(* PLC project marvel_dome, Institute of Astronomy Onto 0.0.1 *)
(* stored: creationDateTime 2025-02-14T19:08:53.030329, modificationDateTime 2025-02-14T19:08:53.030329 *)

TYPE DomeShutterMotionStates : (STANDSTILL := 0, OPENING := 1, CLOSING := 2, STOPPING := 3, TIMEOUT_ERROR := 4, RETRY_OPENING := 5, RETRY_CLOSING := 6, UNKNOWN_DRIVE_LOGIC_ERROR := 7) BYTE;
END_TYPE

TYPE DomeShutterApertureStates : (UNKNOWN := 0, FULLY_OPEN := 1, PARTIALLY_OPEN := 2, FULLY_CLOSED := 3, INVALID := 4) BYTE;
END_TYPE

TYPE DomeShutterCommands : (NONE := 0, STOP := 1, CLOSE := 2, OPEN := 3, SET_HUMIDITY_LIMIT := 4, SET_HEARTBEAT_TIMEOUT := 5, SET_DRIVE_LOGIC := 6) BYTE;
END_TYPE

TYPE DomeShutterDriveLogic : (UNKNOWN := 0, EDGE_BASED := 1, LEVEL_BASED := 2) BYTE;
END_TYPE

TYPE DomeParts : STRUCT
  shutter : DomeShutter;  (* Shutter mechanism *)
  rotation : DomeRotation;  (* Rotation mechanism *)
END_STRUCT;
END_TYPE

TYPE DomeRotationParts : STRUCT
  motorAxis : AngularAxis;  (* Motor axis *)
  encoderAxis : AngularAxis;  (* Encoder axis *)
END_STRUCT;
END_TYPE

TYPE DomeProcesses : STRUCT
  initialize : Process;  (* Start initializing *)
  changeOperatingState : ChangeOperatingStateProcess;  (* Change the operating state (e.g. AUTO, MANUAL, ...) *)
  lock : Process;  (* Lock the cover *)
  unlock : Process;  (* Unlock the cover *)
  reset : Process;  (* Reset any errors *)
  powerOn : Process;  (* Power on the dome *)
  powerOff : Process;  (* Power off the dome *)
  syncWithAxes : Process;  (* Synchronize the dome once with the axes *)
  startTracking : Process;  (* Start tracking the axes *)
  stopTracking : Process;  (* Stop tracking the axes *)
  stop : Process;  (* Stop the rotation movement and/or tracking *)
  moveKnownPosition : DomeMoveKnownPositionProcess;  (* Move the dome to the given known position *)
END_STRUCT;
END_TYPE

TYPE DomeShutterProcesses : STRUCT
  open : Process;  (* Open both panels *)
  close : Process;  (* Close both panels *)
  stop : Process;  (* Stop the panels *)
END_STRUCT;
END_TYPE

TYPE DomeRotationProcesses : STRUCT
  reset : Process;  (* Reset errors *)
  stop : Process;  (* Stop the rotation *)
  moveAbsolute : DomeMoveProcess;  (* Move absolute *)
  moveRelative : DomeMoveProcess;  (* Move relative *)
  powerOn : Process;  (* Power on master and slave *)
  powerOff : Process;  (* Power off master and slave *)
END_STRUCT;
END_TYPE

TYPE DomeStatuses : STRUCT
  initializationStatus : InitializationStatus;
  healthStatus : HealthStatus;
  busyStatus : BusyStatus;
  operatingStatus : OperatingStatus;
  poweredStatus : PoweredStatus;
END_STRUCT;
END_TYPE

TYPE DomeShutterStatuses : STRUCT
  apertureStatus : ApertureStatus;  (* Combined aperture status (i.e. of both panels) *)
  motionStatus : DomeShutterOpeningStatus;  (* Motion status *)
  healthStatus : HealthStatus;  (* Health status *)
  busyStatus : BusyStatus;  (* Busy status *)
END_STRUCT;
END_TYPE

TYPE DomeRotationStatuses : STRUCT
  healthStatus : HealthStatus;  (* Health status *)
  busyStatus : BusyStatus;  (* Busy status *)
  poweredStatus : PoweredStatus;  (* Powered status *)
END_STRUCT;
END_TYPE

TYPE DomeConfig : STRUCT
  shutter : DomeShutterConfig;  (* The config of the shutter mechanism *)
  rotation : DomeRotationConfig;  (* The config of the rotation system *)
  maxTrackingDistance : LREAL;  (* The maximum distance between telescope and dome while tracking *)
  trackingLoopTime : LREAL;  (* Loop time, in seconds, of the tracking. *)
  knownPositions : DomeKnownPositionsConfig;  (* The known positions of the dome *)
  knownPositionTolerance : LREAL;  (* Tolerance (in degrees) to determine if the dome is at a known position *)
END_STRUCT;
END_TYPE

TYPE DomeKnownPositionConfig : STRUCT
  name : STRING;  (* The name of the position (e.g. 'PARK') *)
  position : LREAL;  (* Azimuth in degrees *)
END_STRUCT;
END_TYPE

TYPE DomeKnownPositionsConfig : STRUCT
  position0 : DomeKnownPositionConfig;  (* Known position 0 *)
  position1 : DomeKnownPositionConfig;  (* Known position 1 *)
  position2 : DomeKnownPositionConfig;  (* Known position 2 *)
  position3 : DomeKnownPositionConfig;  (* Known position 3 *)
  position4 : DomeKnownPositionConfig;  (* Known position 4 *)
  position5 : DomeKnownPositionConfig;  (* Known position 5 *)
  position6 : DomeKnownPositionConfig;  (* Known position 6 *)
  position7 : DomeKnownPositionConfig;  (* Known position 7 *)
  position8 : DomeKnownPositionConfig;  (* Known position 8 *)
  position9 : DomeKnownPositionConfig;  (* Known position 9 *)
END_STRUCT;
END_TYPE

TYPE DomeShutterConfig : STRUCT
  remotePlcAmsId : STRING;  (* AMS ID of the shutter PLC *)
  remotePlcTimeoutSeconds : LREAL;  (* The timeout of a single ADS command. *)
  simulated : BOOL := TRUE;  (* TRUE if the shutter is simulated, FALSE if not *)
  openingTimeoutSeconds : LREAL;  (* The opening timeout. *)
  closingTimeoutSeconds : LREAL;  (* The closing timeout. *)
END_STRUCT;
END_TYPE

TYPE DomeRotationConfig : STRUCT
  maxMovingVelocity : LREAL;  (* Maximum velocity when moving absolute or relative, in degrees per second *)
  maxMasterSlaveLag : LREAL;  (* Below this lag value (in degrees), the lag is considered not an error *)
  homePosition : LREAL;  (* Azimuth position of the home sensor, in degrees *)
END_STRUCT;
END_TYPE

{attribute 'pack_mode' := '8'}
TYPE DomeShutterDataRead : STRUCT
  motionState : DomeShutterMotionStates;  (* The motion state, as reported by the shutter PLC *)
  apertureState : DomeShutterApertureStates;  (* The aperture state, as reported by the shutter PLC *)
  heartBeatReceived : UDINT;  (* The heartbeat that was last received by the shutter PLC, as reported by the shutter PLC *)
  lastCommandReceived : DomeShutterCommands;  (* The command that was last received by the shutter PLC, as reported by the shutter PLC *)
  leftPanelOpen : BIT;  (* True if the left panel is open, False if not *)
  leftPanelClosed : BIT;  (* True if the left panel is closed, False if not *)
  rightPanelOpen : BIT;  (* True if the right panel is open, False if not *)
  rightPanelClosed : BIT;  (* True if the right panel is closed, False if not *)
  relayOpenActive : BIT;  (* True if the relay to open the shutter is active, False if not *)
  relayCloseActive : BIT;  (* True if the relay to close the shutter is active, False if not *)
  bHumidityUnderrange : BIT;  (* True if the humidity sensor is in underrange, False if not *)
  bHumidityOverrange : BIT;  (* True if the humidity sensor is in overrange, False if not *)
  bHumidityError : BIT;  (* True if the humidity sensor is in error, False if not *)
  bTemperatureUnderrange : BIT;  (* True if the temperature sensor is in underrange, False if not *)
  bTemperatureOverrange : BIT;  (* True if the temperature sensor is in overrange, False if not *)
  bTemperatureError : BIT;  (* True if the temperature sensor is in error, False if not *)
  heartBeatViolation : BIT;  (* True if there is a missing heartbeat reported by the shutter PLC, False if not *)
  humidityViolation : BIT;  (* True if there is high humidity reported by the shutter PLC, False if not *)
  driveLogic : DomeShutterDriveLogic;  (* Determines which logic is used by the shutter drives (edge or level based) *)
  humidityRawValue : INT;  (* The raw value of the humidity sensor *)
  temperatureRawValue : INT;  (* The raw value of the temperature sensor *)
  humidityLimit : INT;  (* Humidity limit (as raw sensor value) above which the dome will close automatically (-1 means turn off) *)
  heartBeatTimeout : INT;  (* Heartbeat timeout (in seconds) above which the dome will close automatically (-1 means turn off) *)
END_STRUCT;
END_TYPE

{attribute 'pack_mode' := '8'}
TYPE DomeShutterDataWrite : STRUCT
  heartBeat : UDINT;  (* The heartbeat to send to the shutter PLC *)
  command : DomeShutterCommands;  (* The command to send to the shutter PLC *)
  arg : INT;  (* The int16 argument belonging to the command (optional) *)
END_STRUCT;
END_TYPE

TYPE DomeMoveKnownPositionProcessArgs : STRUCT
  name : STRING;  (* Name of the position to move to *)
END_STRUCT;
END_TYPE

TYPE DomeMoveProcessArgs : STRUCT
  position : LREAL;  (* New absolute or relative position value in degrees *)
END_STRUCT;
END_TYPE

FUNCTION_BLOCK DomeShutterOpeningStatus
  VAR_INPUT
    superState : BOOL := TRUE;  (* Super state (TRUE if the super state is active, or if there is no super state) *)
    shutterValue : DomeShutterMotionStates;  (* Enum from mini PLC *)
  END_VAR
  VAR_OUTPUT
    {attribute 'OPC.UA.DA' := '1'}
    {attribute 'OPC.UA.DA.Access' := '1'}
    standstill : BOOL;  (* Standstill *)
    {attribute 'OPC.UA.DA' := '1'}
    {attribute 'OPC.UA.DA.Access' := '1'}
    opening : BOOL;  (* Opening *)
    {attribute 'OPC.UA.DA' := '1'}
    {attribute 'OPC.UA.DA.Access' := '1'}
    closing : BOOL;  (* Closing *)
    {attribute 'OPC.UA.DA' := '1'}
    {attribute 'OPC.UA.DA.Access' := '1'}
    stopping : BOOL;  (* Stopping *)
    {attribute 'OPC.UA.DA' := '1'}
    {attribute 'OPC.UA.DA.Access' := '1'}
    timeoutError : BOOL;  (* Timeout error *)
    {attribute 'OPC.UA.DA' := '1'}
    {attribute 'OPC.UA.DA.Access' := '1'}
    retryOpening : BOOL;  (* Retry opening *)
    {attribute 'OPC.UA.DA' := '1'}
    {attribute 'OPC.UA.DA.Access' := '1'}
    retryClosing : BOOL;  (* Retry closing *)
    {attribute 'OPC.UA.DA' := '1'}
    {attribute 'OPC.UA.DA.Access' := '1'}
    unknownDriveLogicError : BOOL;  (* Drive logic (edge based or dead-man switch) was not configured yet *)
  END_VAR

            standstill := (shutterValue = DomeShutterMotionStates.STANDSTILL) AND superState;
opening := (shutterValue = DomeShutterMotionStates.OPENING) AND superState;
closing := (shutterValue = DomeShutterMotionStates.CLOSING) AND superState;
stopping := (shutterValue = DomeShutterMotionStates.STOPPING) AND superState;
timeoutError := (shutterValue = DomeShutterMotionStates.TIMEOUT_ERROR) AND superState;
retryOpening := (shutterValue = DomeShutterMotionStates.RETRY_OPENING) AND superState;
retryClosing := (shutterValue = DomeShutterMotionStates.RETRY_CLOSING) AND superState;
unknownDriveLogicError := (shutterValue = DomeShutterMotionStates.UNKNOWN_DRIVE_LOGIC_ERROR) AND superState;

          
END_FUNCTION_BLOCK

FUNCTION_BLOCK SM_Dome
  VAR_OUTPUT
    {attribute 'OPC.UA.DA' := '1'}
    {attribute 'OPC.UA.DA.Access' := '1'}
    actualStatus : STRING;  (* Current status description *)
    previousStatus : STRING;  (* Previous status description *)
    {attribute 'OPC.UA.DA' := '1'}
    {attribute 'OPC.UA.DA.Access' := '1'}
    isTracking : BOOL;  (* True if the dome is tracking the telescope *)
    {attribute 'OPC.UA.DA' := '1'}
    {attribute 'OPC.UA.DA.Access' := '1'}
    isAtKnownPosition : BOOL;  (* True if the dome is at a known position *)
    {attribute 'OPC.UA.DA' := '1'}
    {attribute 'OPC.UA.DA.Access' := '1'}
    actualKnownPositionName : STRING;  (* Name of the known position if isAtKnownPosition is True *)
    statuses : DomeStatuses;  (* Statuses of the state machine *)
    parts : DomeParts;  (* Parts of the state machine *)
    processes : DomeProcesses;  (* Processes of the state machine *)
  END_VAR
  VAR_IN_OUT
    {attribute 'OPC.UA.DA' := '0'}
    operatorStatus : OperatorStatus;  (* Reference to the operator (observer/tech) *)
    {attribute 'OPC.UA.DA' := '0'}
    activityStatus : ActivityStatus;  (* Shared activity status *)
    {attribute 'OPC.UA.DA' := '0'}
    config : DomeConfig;  (* Active configuration of the cover *)
    {attribute 'OPC.UA.DA' := '0'}
    telescopeAzi : AngularPosition;  (* Azimuth target position of the telescope Axes *)
  END_VAR

            parts.shutter(
    initializationStatus := statuses.initializationStatus,
    operatorStatus := operatorStatus,
    operatingStatus := statuses.operatingStatus,
    activityStatus := activityStatus,
    config := config.shutter);
parts.rotation(
    initializationStatus := statuses.initializationStatus,
    operatorStatus := operatorStatus,
    operatingStatus := statuses.operatingStatus,
    config := config.rotation);
statuses.initializationStatus();
statuses.healthStatus(
    isGood := parts.shutter.statuses.healthStatus.isGood AND parts.rotation.statuses.healthStatus.isGood,
    hasWarning := parts.shutter.statuses.healthStatus.hasWarning OR parts.rotation.statuses.healthStatus.hasWarning);
statuses.busyStatus( isBusy := parts.shutter.statuses.busyStatus.busy OR parts.rotation.statuses.busyStatus.busy );
statuses.operatingStatus( superState := statuses.initializationStatus.initialized );
statuses.poweredStatus( isEnabled := parts.rotation.statuses.poweredStatus.enabled );
processes.initialize( isEnabled := (NOT(statuses.initializationStatus.locked)) AND (statuses.initializationStatus.shutdown OR (statuses.initializationStatus.initializingFailed OR statuses.initializationStatus.initialized)) );
processes.changeOperatingState( isEnabled := FALSE );
processes.lock( isEnabled := operatorStatus.tech );
processes.unlock( isEnabled := operatorStatus.tech AND statuses.initializationStatus.locked );
processes.reset( isEnabled := statuses.busyStatus.idle AND statuses.initializationStatus.initialized );
processes.powerOn( isEnabled := (NOT(statuses.initializationStatus.locked)) AND (statuses.initializationStatus.initialized AND processes.powerOn.statuses.busyStatus.idle) );
processes.powerOff( isEnabled := statuses.initializationStatus.initialized AND processes.powerOff.statuses.busyStatus.idle );
processes.syncWithAxes( isEnabled := statuses.initializationStatus.initialized AND (statuses.busyStatus.idle AND statuses.poweredStatus.enabled) );
processes.startTracking( isEnabled := statuses.poweredStatus.enabled AND (NOT(isTracking)) );
processes.stopTracking( isEnabled := isTracking );
processes.stop( isEnabled := statuses.busyStatus.busy OR (isTracking OR operatorStatus.tech) );
processes.moveKnownPosition( isEnabled := statuses.initializationStatus.initialized AND (statuses.busyStatus.idle AND statuses.poweredStatus.enabled) );

          

{attribute 'TcRpcEnable' := '1'}
METHOD initialize : RequestResults
                  initialize := THIS^.processes.initialize.request();

                
END_METHOD

{attribute 'TcRpcEnable' := '1'}
METHOD changeOperatingState : RequestResults
  VAR_INPUT
    state : OperatingStates;
  END_VAR
                  changeOperatingState := THIS^.processes.changeOperatingState.request( state := state );

                
END_METHOD

{attribute 'TcRpcEnable' := '1'}
METHOD lock : RequestResults
                  lock := THIS^.processes.lock.request();

                
END_METHOD

{attribute 'TcRpcEnable' := '1'}
METHOD unlock : RequestResults
                  unlock := THIS^.processes.unlock.request();

                
END_METHOD

{attribute 'TcRpcEnable' := '1'}
METHOD reset : RequestResults
                  reset := THIS^.processes.reset.request();

                
END_METHOD

{attribute 'TcRpcEnable' := '1'}
METHOD powerOn : RequestResults
                  powerOn := THIS^.processes.powerOn.request();

                
END_METHOD

{attribute 'TcRpcEnable' := '1'}
METHOD powerOff : RequestResults
                  powerOff := THIS^.processes.powerOff.request();

                
END_METHOD

{attribute 'TcRpcEnable' := '1'}
METHOD syncWithAxes : RequestResults
                  syncWithAxes := THIS^.processes.syncWithAxes.request();

                
END_METHOD

{attribute 'TcRpcEnable' := '1'}
METHOD startTracking : RequestResults
                  startTracking := THIS^.processes.startTracking.request();

                
END_METHOD

{attribute 'TcRpcEnable' := '1'}
METHOD stopTracking : RequestResults
                  stopTracking := THIS^.processes.stopTracking.request();

                
END_METHOD

{attribute 'TcRpcEnable' := '1'}
METHOD stop : RequestResults
                  stop := THIS^.processes.stop.request();

                
END_METHOD

{attribute 'TcRpcEnable' := '1'}
METHOD moveKnownPosition : RequestResults
  VAR_INPUT
    name : STRING;
  END_VAR
                  moveKnownPosition := THIS^.processes.moveKnownPosition.request( name := name );

                
END_METHOD

METHOD _log : BOOL
  VAR_INPUT
    name : STRING;  (* Name of this function block instance *)
  END_VAR
  VAR_IN_OUT
    buffer : LogBuffer;  (* Buffer to write all logging to *)
  END_VAR
  VAR
    subBuffer : LogBuffer;  (* Temporary buffer to write logging by parts (sub-statemachines) to *)
  END_VAR
                  THIS^.parts.shutter._log(
    name := 'shutter',
    buffer := subBuffer);
THIS^.parts.rotation._log(
    name := 'rotation',
    buffer := subBuffer);
THIS^.processes.initialize._log(
    name := 'processes.initialize',
    buffer := subBuffer);
THIS^.processes.changeOperatingState._log(
    name := 'processes.changeOperatingState',
    buffer := subBuffer);
THIS^.processes.lock._log(
    name := 'processes.lock',
    buffer := subBuffer);
THIS^.processes.unlock._log(
    name := 'processes.unlock',
    buffer := subBuffer);
THIS^.processes.reset._log(
    name := 'processes.reset',
    buffer := subBuffer);
THIS^.processes.powerOn._log(
    name := 'processes.powerOn',
    buffer := subBuffer);
THIS^.processes.powerOff._log(
    name := 'processes.powerOff',
    buffer := subBuffer);
THIS^.processes.syncWithAxes._log(
    name := 'processes.syncWithAxes',
    buffer := subBuffer);
THIS^.processes.startTracking._log(
    name := 'processes.startTracking',
    buffer := subBuffer);
THIS^.processes.stopTracking._log(
    name := 'processes.stopTracking',
    buffer := subBuffer);
THIS^.processes.stop._log(
    name := 'processes.stop',
    buffer := subBuffer);
THIS^.processes.moveKnownPosition._log(
    name := 'processes.moveKnownPosition',
    buffer := subBuffer);
LOGGER(
    name := name,
    actualStatus := THIS^.actualStatus,
    previousStatus := THIS^.previousStatus,
    buffer := buffer,
    subBuffer := subBuffer,
    pHealthStatus := ADR(THIS^.statuses.healthStatus),
    pBusyStatus := ADR(THIS^.statuses.busyStatus));

                
END_METHOD
END_FUNCTION_BLOCK

FUNCTION_BLOCK SM_DomeShutter
  VAR_INPUT
    {attribute 'OPC.UA.DA' := '1'}
    {attribute 'OPC.UA.DA.Access' := '1'}
    dataRead : DomeShutterDataRead;  (* The data read from the shutter PLC via Bluetooth *)
    {attribute 'OPC.UA.DA' := '1'}
    {attribute 'OPC.UA.DA.Access' := '1'}
    dataWrite : DomeShutterDataWrite;  (* The data written to the shutter PLC via Bluetooth *)
    {attribute 'OPC.UA.DA' := '1'}
    {attribute 'OPC.UA.DA.Access' := '1'}
    adsReadError : BOOL;  (* True if the ADS Read communication to the shutter PLC is in error *)
    {attribute 'OPC.UA.DA' := '1'}
    {attribute 'OPC.UA.DA.Access' := '1'}
    adsReadErrorId : UDINT;  (* The error id if adsReadError is true *)
    {attribute 'OPC.UA.DA' := '1'}
    {attribute 'OPC.UA.DA.Access' := '1'}
    adsWriteError : BOOL;  (* True if the ADS Read communication to the shutter PLC is in error *)
    {attribute 'OPC.UA.DA' := '1'}
    {attribute 'OPC.UA.DA.Access' := '1'}
    adsWriteErrorId : UDINT;  (* The error id if adsReadError is true *)
  END_VAR
  VAR_OUTPUT
    {attribute 'OPC.UA.DA' := '1'}
    {attribute 'OPC.UA.DA.Access' := '1'}
    actualStatus : STRING;  (* Current status description *)
    previousStatus : STRING;  (* Previous status description *)
    {attribute 'OPC.UA.DA' := '1'}
    {attribute 'OPC.UA.DA.Access' := '1'}
    isSimulated : BOOL;  (* True if the shutter is being simulated *)
    {attribute 'OPC.UA.DA' := '1'}
    {attribute 'OPC.UA.DA.Access' := '1'}
    isConnected : BOOL;  (* True if the shutter PLC is connected *)
    statuses : DomeShutterStatuses;  (* Statuses of the state machine *)
    processes : DomeShutterProcesses;  (* Processes of the state machine *)
  END_VAR
  VAR_IN_OUT
    {attribute 'OPC.UA.DA' := '0'}
    initializationStatus : InitializationStatus;  (* Dome initialization status (initialized/initializing/...) *)
    {attribute 'OPC.UA.DA' := '0'}
    operatorStatus : OperatorStatus;  (* MTCS operator (observer/tech) *)
    {attribute 'OPC.UA.DA' := '0'}
    operatingStatus : OperatingStatus;  (* Dome operating status (manual/auto) *)
    {attribute 'OPC.UA.DA' := '0'}
    activityStatus : ActivityStatus;  (* Shared activity status *)
    {attribute 'OPC.UA.DA' := '0'}
    config : DomeShutterConfig;  (* The shutter config *)
  END_VAR

            statuses.apertureStatus(
    superState := NOT((dataRead.apertureState = DomeShutterApertureStates.UNKNOWN) OR (dataRead.apertureState = DomeShutterApertureStates.INVALID)),
    isOpen := dataRead.apertureState = DomeShutterApertureStates.FULLY_OPEN,
    isClosed := dataRead.apertureState = DomeShutterApertureStates.FULLY_CLOSED);
statuses.motionStatus( shutterValue := dataRead.motionState );
statuses.healthStatus(
    superState := NOT(initializationStatus.shutdown),
    isGood := isConnected AND (processes.open.statuses.healthStatus.isGood AND (processes.close.statuses.healthStatus.isGood AND processes.stop.statuses.healthStatus.isGood)),
    hasWarning := (processes.open.statuses.healthStatus.hasWarning OR (processes.close.statuses.healthStatus.hasWarning OR processes.stop.statuses.healthStatus.hasWarning)) OR (statuses.busyStatus.idle AND statuses.apertureStatus.partiallyOpen));
statuses.busyStatus(
    superState := NOT(initializationStatus.shutdown),
    isBusy := processes.open.statuses.busyStatus.busy OR (processes.close.statuses.busyStatus.busy OR processes.stop.statuses.busyStatus.busy));
processes.open( isEnabled := statuses.healthStatus.isGood AND ((NOT(initializationStatus.locked)) AND (operatorStatus.tech OR (statuses.busyStatus.idle AND (initializationStatus.initialized AND (activityStatus.awake OR activityStatus.moving))))) );
processes.close( isEnabled := operatorStatus.tech OR (statuses.healthStatus.isGood AND ((NOT(initializationStatus.locked)) AND (statuses.busyStatus.idle AND initializationStatus.initialized))) );
processes.stop( isEnabled := statuses.busyStatus.busy );

          

{attribute 'TcRpcEnable' := '1'}
METHOD open : RequestResults
                  open := THIS^.processes.open.request();

                
END_METHOD

{attribute 'TcRpcEnable' := '1'}
METHOD close : RequestResults
                  close := THIS^.processes.close.request();

                
END_METHOD

{attribute 'TcRpcEnable' := '1'}
METHOD stop : RequestResults
                  stop := THIS^.processes.stop.request();

                
END_METHOD

METHOD _log : BOOL
  VAR_INPUT
    name : STRING;  (* Name of this function block instance *)
  END_VAR
  VAR_IN_OUT
    buffer : LogBuffer;  (* Buffer to write all logging to *)
  END_VAR
  VAR
    subBuffer : LogBuffer;  (* Temporary buffer to write logging by parts (sub-statemachines) to *)
  END_VAR
                  THIS^.processes.open._log(
    name := 'processes.open',
    buffer := subBuffer);
THIS^.processes.close._log(
    name := 'processes.close',
    buffer := subBuffer);
THIS^.processes.stop._log(
    name := 'processes.stop',
    buffer := subBuffer);
LOGGER(
    name := name,
    actualStatus := THIS^.actualStatus,
    previousStatus := THIS^.previousStatus,
    buffer := buffer,
    subBuffer := subBuffer,
    pHealthStatus := ADR(THIS^.statuses.healthStatus),
    pBusyStatus := ADR(THIS^.statuses.busyStatus));

                
END_METHOD
END_FUNCTION_BLOCK

FUNCTION_BLOCK SM_DomeRotation
  VAR_OUTPUT
    {attribute 'OPC.UA.DA' := '1'}
    {attribute 'OPC.UA.DA.Access' := '1'}
    actualStatus : STRING;  (* Current status description *)
    previousStatus : STRING;  (* Previous status description *)
    {attribute 'OPC.UA.DA' := '1'}
    {attribute 'OPC.UA.DA.Access' := '1'}
    actPos : AngularPosition;  (* The actual position (same as parts.masterAxis!) *)
    {attribute 'OPC.UA.DA' := '1'}
    {attribute 'OPC.UA.DA.Access' := '1'}
    actVelo : AngularVelocity;  (* The actual velocity (same as parts.masterAxis!) *)
    statuses : DomeRotationStatuses;  (* Statuses of the state machine *)
    parts : DomeRotationParts;  (* Parts of the state machine *)
    processes : DomeRotationProcesses;  (* Processes of the state machine *)
  END_VAR
  VAR_IN_OUT
    {attribute 'OPC.UA.DA' := '0'}
    initializationStatus : InitializationStatus;  (* Reference to the MTCS initialization status *)
    {attribute 'OPC.UA.DA' := '0'}
    operatorStatus : OperatorStatus;  (* Reference to the MTCS operator status *)
    {attribute 'OPC.UA.DA' := '0'}
    operatingStatus : OperatingStatus;  (* Reference to the Dome operating status *)
    {attribute 'OPC.UA.DA' := '0'}
    config : DomeRotationConfig;  (* Reference to the rotation config *)
  END_VAR

            parts.motorAxis( isEnabled := (NOT(initializationStatus.locked)) AND operatorStatus.tech );
parts.encoderAxis( isEnabled := (NOT(initializationStatus.locked)) AND operatorStatus.tech );
statuses.healthStatus(
    isGood := parts.motorAxis.statuses.healthStatus.isGood AND (parts.encoderAxis.statuses.healthStatus.isGood AND (processes.reset.statuses.healthStatus.isGood AND processes.stop.statuses.healthStatus.isGood)),
    hasWarning := parts.motorAxis.statuses.healthStatus.hasWarning OR (parts.encoderAxis.statuses.healthStatus.hasWarning OR (processes.reset.statuses.healthStatus.hasWarning OR processes.stop.statuses.healthStatus.hasWarning)));
statuses.busyStatus( isBusy := parts.motorAxis.statuses.busyStatus.busy OR (parts.encoderAxis.statuses.busyStatus.busy OR (processes.reset.statuses.busyStatus.busy OR processes.stop.statuses.busyStatus.busy)) );
statuses.poweredStatus( isEnabled := parts.motorAxis.statuses.poweredStatus.enabled );
processes.reset( isEnabled := statuses.busyStatus.idle );
processes.stop( isEnabled := statuses.busyStatus.busy OR operatorStatus.tech );
processes.moveAbsolute( isEnabled := statuses.busyStatus.idle AND statuses.poweredStatus.enabled );
processes.moveRelative( isEnabled := processes.moveAbsolute.isEnabled );
processes.powerOn( isEnabled := (NOT(initializationStatus.locked)) AND statuses.busyStatus.idle );
processes.powerOff( isEnabled := statuses.busyStatus.idle );

          

{attribute 'TcRpcEnable' := '1'}
METHOD reset : RequestResults
                  reset := THIS^.processes.reset.request();

                
END_METHOD

{attribute 'TcRpcEnable' := '1'}
METHOD stop : RequestResults
                  stop := THIS^.processes.stop.request();

                
END_METHOD

{attribute 'TcRpcEnable' := '1'}
METHOD moveAbsolute : RequestResults
  VAR_INPUT
    position : LREAL;
  END_VAR
                  moveAbsolute := THIS^.processes.moveAbsolute.request( position := position );

                
END_METHOD

{attribute 'TcRpcEnable' := '1'}
METHOD moveRelative : RequestResults
  VAR_INPUT
    position : LREAL;
  END_VAR
                  moveRelative := THIS^.processes.moveRelative.request( position := position );

                
END_METHOD

{attribute 'TcRpcEnable' := '1'}
METHOD powerOn : RequestResults
                  powerOn := THIS^.processes.powerOn.request();

                
END_METHOD

{attribute 'TcRpcEnable' := '1'}
METHOD powerOff : RequestResults
                  powerOff := THIS^.processes.powerOff.request();

                
END_METHOD

METHOD _log : BOOL
  VAR_INPUT
    name : STRING;  (* Name of this function block instance *)
  END_VAR
  VAR_IN_OUT
    buffer : LogBuffer;  (* Buffer to write all logging to *)
  END_VAR
  VAR
    subBuffer : LogBuffer;  (* Temporary buffer to write logging by parts (sub-statemachines) to *)
  END_VAR
                  THIS^.parts.motorAxis._log(
    name := 'motorAxis',
    buffer := subBuffer);
THIS^.parts.encoderAxis._log(
    name := 'encoderAxis',
    buffer := subBuffer);
THIS^.processes.reset._log(
    name := 'processes.reset',
    buffer := subBuffer);
THIS^.processes.stop._log(
    name := 'processes.stop',
    buffer := subBuffer);
THIS^.processes.moveAbsolute._log(
    name := 'processes.moveAbsolute',
    buffer := subBuffer);
THIS^.processes.moveRelative._log(
    name := 'processes.moveRelative',
    buffer := subBuffer);
THIS^.processes.powerOn._log(
    name := 'processes.powerOn',
    buffer := subBuffer);
THIS^.processes.powerOff._log(
    name := 'processes.powerOff',
    buffer := subBuffer);
LOGGER(
    name := name,
    actualStatus := THIS^.actualStatus,
    previousStatus := THIS^.previousStatus,
    buffer := buffer,
    subBuffer := subBuffer,
    pHealthStatus := ADR(THIS^.statuses.healthStatus),
    pBusyStatus := ADR(THIS^.statuses.busyStatus));

                
END_METHOD
END_FUNCTION_BLOCK

FUNCTION_BLOCK DomeMoveKnownPositionProcess EXTENDS BaseProcess
  VAR_INPUT
    {attribute 'OPC.UA.DA' := '1'}
    set : DomeMoveKnownPositionProcessArgs;  (* Arguments to be set, before writing do_request TRUE *)
  END_VAR
  VAR_OUTPUT
    {attribute 'OPC.UA.DA' := '1'}
    {attribute 'OPC.UA.DA.Access' := '1'}
    get : DomeMoveKnownPositionProcessArgs;  (* Arguments in use by the process, if do_request was accepted *)
  END_VAR

            IF do_request THEN
    do_request_result := request( name := set.name );
    do_request := FALSE;
END_IF;
SUPER^();

          

{attribute 'TcRpcEnable' := '1'}
METHOD start
  VAR_INPUT
    name : STRING;  (* Name of the position to move to *)
  END_VAR
                  THIS^.get.name := name;
THIS^.statuses.busyStatus( isBusy := TRUE );
THIS^.statuses.healthStatus( isGood := TRUE );

                
END_METHOD

{attribute 'TcRpcEnable' := '1'}
METHOD request : RequestResults
  VAR_INPUT
    name : STRING;  (* Name of the position to move to *)
  END_VAR
                  IF THIS^.statuses.enabledStatus.enabled THEN
    request := RequestResults.ACCEPTED;
    THIS^.start( name := name );
ELSE
    request := RequestResults.REJECTED;
END_IF;

                
END_METHOD
END_FUNCTION_BLOCK

FUNCTION_BLOCK DomeMoveProcess EXTENDS BaseProcess
  VAR_INPUT
    {attribute 'OPC.UA.DA' := '1'}
    set : DomeMoveProcessArgs;  (* Arguments to be set, before writing do_request TRUE *)
  END_VAR
  VAR_OUTPUT
    {attribute 'OPC.UA.DA' := '1'}
    {attribute 'OPC.UA.DA.Access' := '1'}
    get : DomeMoveProcessArgs;  (* Arguments in use by the process, if do_request was accepted *)
  END_VAR

            IF do_request THEN
    do_request_result := request( position := set.position );
    do_request := FALSE;
END_IF;
SUPER^();

          

{attribute 'TcRpcEnable' := '1'}
METHOD start
  VAR_INPUT
    position : LREAL;  (* New absolute or relative position value in degrees *)
  END_VAR
                  THIS^.get.position := position;
THIS^.statuses.busyStatus( isBusy := TRUE );
THIS^.statuses.healthStatus( isGood := TRUE );

                
END_METHOD

{attribute 'TcRpcEnable' := '1'}
METHOD request : RequestResults
  VAR_INPUT
    position : LREAL;  (* New absolute or relative position value in degrees *)
  END_VAR
                  IF THIS^.statuses.enabledStatus.enabled THEN
    request := RequestResults.ACCEPTED;
    THIS^.start( position := position );
ELSE
    request := RequestResults.REJECTED;
END_IF;

                
END_METHOD
END_FUNCTION_BLOCK
